Universal Robots PolyScope program: seek_with_force.urp

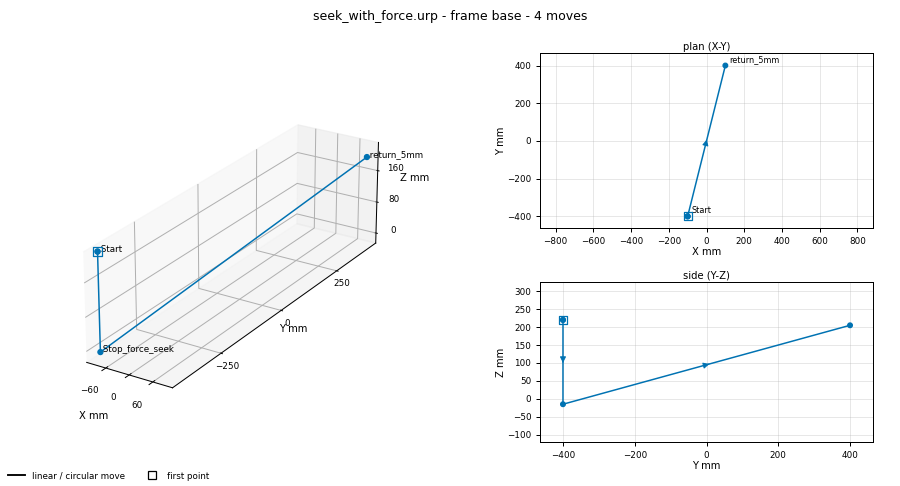
[picture p0: tool path of seek_with_force.urp in frame base, 4 of 4 moves have a stored position in this frame; points joined in program order, loops and branches not executed]
ProgramRoot directory=/home/ur/ursim-3.1/programs/Support site; kinematics=(a=[0.00008, -0.27626, -0.39154, 0.00008, -0.00003, 0], d=[0.08934, 419.16584, -412.94914, -6.10665, 0.09493, 0.08212], alpha=[1.57022, 0.00077, -0.00486, 1.57064, -1.57023, 0], deltaTheta=[-0.00002, 0.86369, -0.94076, 0.07711, 0.00006, 0], status=notLinearised); lastSavedInVersion=(project__name=Polyscope, major__version=3, minor__version=1, svn__revision=18024, build__date=Jul 07 2015, 15:18:49); name=seek_with_force; programVersion=(project__name=Polyscope, major__version=3, minor__version=1, svn__revision=18024, build__date=Jul 07 2015, 15:18:49); robotEnvironmentFileName=default; serialNumberRobot=2015350001
  BeforeStart description=COMMAND_SEQUENCE_BEFORE_PROGRAM_START; name=BeforeStart
    Move cartesianAcceleration=1.2; cartesianSpeed=0.25; jointAcceleration=1.3962634015954636; jointSpeed=1.0471975511965976; sharedProcessMoveBlendRadius=0.025; motionType=JOINT_SPACE
      Waypoint blendRadius=0.05; cartesianAcceleration=1.2; cartesianSpeed=0.25; jointAcceleration=1.3962634015954636; jointSpeed=1.0471975511965976; nextMotionTime=2.0; stoppoint=true; useSharedBlendParameter=true; useSharedParameters=true; position=TCP in base x=-100.03 y=-399.985 z=220 mm, rx=0.0001 ry=3.1399 rz=0.0001 rad; joints [-88.578, -78.615, -111.599, -79.821, 89.816, 1.322] deg; positionType=FIXED_POSITION; waypointPoseInFeatureCoordinates=(pos=(x=-0.10002955831737015, y=-0.39998524849903616, z=0.22), rot=(x=5.127146917425072E-5, y=3.1399356062822212, z=7.591526070898125E-5)); name=Start
  MainProgram cartesianAcceleration=1.2; cartesianSpeed=0.25; jointAcceleration=1.3962634015954636; jointSpeed=1.0471975511965976; sharedProcessMoveBlendRadius=0.025; motionType=JOINT_SPACE
    Wait 
    Move cartesianAcceleration=0.4; cartesianSpeed=0.075; jointAcceleration=1.3962634015954636; jointSpeed=1.0471975511965976; sharedProcessMoveBlendRadius=0.025; motionType=CARTESIAN_SPACE
      Waypoint blendRadius=0.05; cartesianAcceleration=1.2; cartesianSpeed=0.25; jointAcceleration=1.3962634015954636; jointSpeed=1.0471975511965976; nextMotionTime=2.0; stoppoint=true; useSharedBlendParameter=true; useSharedParameters=true; outputFlangePose=(pos=(x=-0.10025160248426901, y=-0.3999917243815475, z=0.3539998158846689), rot=(x=5.12714775009525E-5, y=3.1399356063434594, z=7.591526728947454E-5)); position=TCP in base x=-100.065 y=-399.98 z=219.985 mm, rx=0.0002 ry=3.14 rz=0.0002 rad; joints [-88.578, -78.615, -111.599, -79.821, 89.816, 1.322] deg; positionType=FIXED_POSITION; waypointPoseInFeatureCoordinates=(pos=(x=-0.10006486768829144, y=-0.39998001848078246, z=0.21998534761552838), rot=(x=1.6862905635080664E-4, y=3.13996773718213, z=1.9039759791381327E-4)); name=Seek_w_force
      If checkConditionInSeperateThread=true; expr=force()<50; type=IF_NODE
        Waypoint blendRadius=0.05; cartesianAcceleration=1.2; cartesianSpeed=0.25; jointAcceleration=1.3962634015954636; jointSpeed=1.0471975511965976; nextMotionTime=2.0; stoppoint=true; useSharedBlendParameter=true; useSharedParameters=true; outputFlangePose=(pos=(x=-0.10024084355344091, y=-0.4000258640752379, z=0.11899987574092918), rot=(x=-1.4688279735575538E-4, y=3.1400657051394867, z=1.4708642955544285E-5)); position=TCP in base x=-100.032 y=-400.036 z=-14.994 mm, rx=-0.0003 ry=3.14 rz=0 rad; joints [-88.531, -98.16, -133.716, -38.157, 89.933, 1.189] deg; positionType=FIXED_POSITION; waypointPoseInFeatureCoordinates=(pos=(x=-0.10003221304994189, y=-0.4000358054743474, z=-0.014993743368692528), rot=(x=-2.812619578391279E-4, y=3.14000220229978, z=1.6934271191152753E-5)); name=Stop_force_seek
      Waypoint blendRadius=0.05; cartesianAcceleration=1.2; cartesianSpeed=0.25; jointAcceleration=1.3962634015954636; jointSpeed=1.0471975511965976; nextMotionTime=2.0; stoppoint=true; useSharedBlendParameter=true; useSharedParameters=true; position=TCP in base x=100 y=400 z=205.001 mm, rx=0 ry=3.14 rz=0 rad; joints [-268.667, -87.663, -127.607, -54.731, 89.909, -178.667] deg; positionType=RELATIVE_POSITION; waypointPoseInFeatureCoordinates=(pos=(x=0.09999998316443576, y=0.40000006613536193, z=0.20500110080726458), rot=(x=-1.647007864217862E-7, y=3.139999996612405, z=5.978965037433122E-7)); name=return_5mm; relativeFromJointPositionVector=(joint=[-4.68912, -1.53871, -2.2346, -0.93912, 1.5692, -3.11832], isUndefined=false); relativeFromToolAxisAngle=(x=-1.6470081565695066E-7, y=3.1399999966120564, z=5.978965037432523E-7); relativeFromToolPosition=(x=0.0999999832782006, y=0.4000000612037796, z=0.20000094556386835)
  Thread name=Thread_1
    Assignment expr=force(); operatorValueType=INTEGER; valueSource=EXPRESSION
    Wait 
